TEXTLIST Mc_Prompts
  0 = 'Machine Prompt 0'
  1 = 'prompt 2'
  2 = 'prompt 3'
   = ''
END_TEXTLIST

(* stored: Version 1.1.0.1, ProductVersion 3.1.4024.12
   TextList Mc_Prompts: Id {503447e5-717e-0dc4-20dd-dba12d898279} *)
